FUNCTION_BLOCK _TOD_TestSuite EXTENDS TcUnit.FB_TestSuite
VAR
END_VAR

TestAddress();
TestClearReference();
TestClone();
TestTypeNameReturnsExpected();
TestMakeReferenceToFollowsReference();
TestMakeReferenceToUpdatesReference();
TestSize();
TestValueReturnsExpectedAfterInit();
TestValueReturnsExpectedAfterChange();
TestSerializeTypeWith();
TestSerializeWith();
TestTryDeserializeFrom();
TestTryMakeReferenceToFollowsReference();
TestTryMakeReferenceToUpdatesReference();

METHOD PUBLIC TestAddress
VAR
    _type : _TOD(TOD#0:0:0);
    notExpected : PVOID := 0;
    actual : PVOID;
END_VAR
TEST('TestAddress');

actual := _type.Address;

AssertFalse(
    Condition := (notExpected = actual),
    Message := 'Type did not return a valid address.'
);

TEST_FINISHED();
END_METHOD

METHOD PUBLIC TestClearReference
VAR
    _type : _TOD(TOD#0:0:0);
	target : TOD := TOD#0:0:0;
    expected : TOD := TOD#0:0:0;
    actual : TOD;
END_VAR
TEST('TestClearReference');

_type.MakeReferenceTo(target);
_type.ClearReference();
target := TOD#12:34:56.789;

actual := _type.Value;

AssertEquals(
    Expected := expected,
    Actual := actual,
    Message := 'Value did not follow target change'
);

TEST_FINISHED();
END_METHOD

METHOD PUBLIC TestClone
VAR
    _type : _TIME_OF_DAY(TIME_OF_DAY#12:34:56.789);
	clone : I_Datatype;
	isValidClone : BOOL;
	compareResult : DINT;
END_VAR
TEST('TestClone');

clone := _type.Clone();

isValidClone := clone <> 0;

IF isValidClone THEN
	compareResult := memcmp(_type.Address, clone.Address, clone.Size);
END_IF

AssertTrue(
	Condition := isValidClone,
	Message := 'Clone did not produce a clone'
);

AssertEquals_DINT(
	Expected := 0,
    Actual := compareResult,
    Message := 'Clone did not return a valid clone.'
);

clone.Dispose();

TEST_FINISHED();
END_METHOD

METHOD PUBLIC TestMakeReferenceToFollowsReference
VAR
    _type : _TOD(TOD#0:0:0);
	target : TOD := TOD#0:0:0;
    expected : TOD := TOD#12:34:56.789;
    actual : TOD;
END_VAR
TEST('TestMakeReferenceToFollowsReference');

_type.MakeReferenceTo(target);
target := TOD#12:34:56.789;

actual := _type.Value;

AssertEquals_TIME_OF_DAY(
    Expected := expected,
    Actual := actual,
    Message := 'Value did not follow target change'
);

TEST_FINISHED();
END_METHOD

METHOD PUBLIC TestMakeReferenceToUpdatesReference
VAR
    _type : _TOD(TOD#0:0:0);
	target : TOD := TOD#0:0:0;
    expected : TOD := TOD#12:34:56.789;
    actual : TOD;
END_VAR
TEST('TestMakeReferenceToUpdatesReference');

_type.MakeReferenceTo(target);
_type.Value := TOD#12:34:56.789;

actual := target;

AssertEquals_TIME_OF_DAY(
    Expected := expected,
    Actual := actual,
    Message := 'Value did not update target'
);

TEST_FINISHED();
END_METHOD

METHOD PUBLIC TestSerializeTypeWith
VAR
    _type : _TOD(TOD#0:0:0);
    serializer : JsonSerializer;
    expected : STRING := '{"typeName":"TOD"}';
    actual : STRING(500);
END_VAR
TEST('TestSerializeTypeWith');

serializer.Reset();
_type.SerializeTypeWith(serializer);
serializer.TryGetSerializedData(ADR(actual), SIZEOF(actual));

AssertEquals_STRING(
    Expected := expected,
    Actual := actual,
    Message := 'Serialization of type did not return correct string.'
);

TEST_FINISHED();
END_METHOD

METHOD PUBLIC TestSerializeWith
VAR
    _type : _TOD(TOD#12:34:56.789);
    serializer : JsonSerializer;
    expected : STRING := '"TOD#12:34:56.789"';
    actual : STRING(500);
END_VAR
TEST('TestSerializeWith');

serializer.Reset();
_type.SerializeWith(serializer);
serializer.TryGetSerializedData(ADR(actual), SIZEOF(actual));

AssertEquals_STRING(
    Expected := expected,
    Actual := actual,
    Message := 'Serialization of type data did not return correct string.'
);

TEST_FINISHED();
END_METHOD

METHOD PUBLIC TestSize
VAR
    _type : _TOD(TOD#0:0:0);
    expected : UDINT := SIZEOF(TOD);
    actual : UDINT;
END_VAR
TEST('TestSize');

actual := _type.Size;

AssertEquals_UDINT(
    Expected := Expected,
    Actual := actual,
    Message := 'Type did not return the correct size.'
);

TEST_FINISHED();
END_METHOD

METHOD PUBLIC TestTryDeserializeFrom
VAR
    deserializer : JsonDeserializer;
    feedback : DeserializerFeedback;
    json : STRING := '"TOD#12:34:56.789"';
    _type : _TOD(TOD#0:0:0);
    expected : TOD := TOD#12:34:56.789;
    actual : TOD;
 END_VAR
TEST('TestTryDeserializeFrom');

deserializer.Reset();
deserializer.TryLoad(json);
_type.TryDeserializeFrom(Deserializer, Feedback);

actual := _type.Value;

AssertEquals_TIME_OF_DAY(
    Expected := expected,
    Actual := actual,
    Message := 'Type did not deserialize correctly.'
);

TEST_FINISHED();
END_METHOD

METHOD PUBLIC TestTryMakeReferenceToFollowsReference
VAR
    _type : _TOD(TOD#0:0:0);
	target : _TOD(TOD#0:0:0);
    expected : TOD := TOD#12:34:56.789;
    actual : TOD;
END_VAR
TEST('TestTryMakeReferenceToFollowsReference');

_type.TryMakeReferenceTo(target);
target.Value := TOD#12:34:56.789;

actual := _type.Value;

AssertEquals_TIME_OF_DAY(
    Expected := expected,
    Actual := actual,
    Message := 'Value did not follow target change'
);

TEST_FINISHED();
END_METHOD

METHOD PUBLIC TestTryMakeReferenceToUpdatesReference
VAR
    _type : _TOD(TOD#0:0:0);
	target : _TOD(TOD#0:0:0);
    expected : TOD := TOD#12:34:56.789;
    actual : TOD;
END_VAR
TEST('TestTryMakeReferenceToUpdatesReference');

_type.TryMakeReferenceTo(target);
_type.Value := TOD#12:34:56.789;

actual := target.Value;

AssertEquals_TIME_OF_DAY(
    Expected := expected,
    Actual := actual,
    Message := 'Value did not update target'
);

TEST_FINISHED();
END_METHOD

METHOD PUBLIC TestTypeNameReturnsExpected
VAR
    _type : _TOD(TOD#0:0:0);
    expected : STRING := 'TOD';
    actual : STRING;
END_VAR
TEST('TestTypeNameReturnsExpected');

actual := _type.TypeName;

AssertEquals_STRING(
    Expected := expected,
    Actual := actual,
    Message := 'Type did not return correct iec type.'
);

TEST_FINISHED();
END_METHOD

METHOD PUBLIC TestValueReturnsExpectedAfterChange
VAR
    _type : _TOD(TOD#0:0:0);
    expected : TOD := TOD#12:34:56.789;
    actual : TOD;
END_VAR
TEST('TestValueReturnsExpectedAfterChange');

_type.Value := TOD#12:34:56.789;

actual := _type.Value;

AssertEquals_TIME_OF_DAY(
    Expected := expected,
    Actual := actual,
    Message := 'Expected value not returned after change.'
);

TEST_FINISHED();
END_METHOD

METHOD PUBLIC TestValueReturnsExpectedAfterInit
VAR
    _type : _TOD(TOD#12:34:56.789);
    expected : TOD := TOD#12:34:56.789;
    actual : TOD;
END_VAR
TEST('TestValueReturnsExpectedAfterInit');

actual := _type.Value;

AssertEquals_TIME_OF_DAY(
    Expected := expected,
    Actual := actual,
    Message := 'Expected value not returned after Init.'
);

TEST_FINISHED();
END_METHOD

END_FUNCTION_BLOCK

(* stored: Version 1.1.0.1, ProductVersion 3.1.4024.12
   POU _TOD_TestSuite: Id {19c985da-db57-4090-99b1-9510d3a8ac67}, SpecialFunc None
   Method TestAddress: Id {498e0ce2-8566-4fad-98f3-21d590e725ad}
   Method TestClearReference: Id {1d1ff48f-8829-450a-ba42-080daad2c195}
   Method TestClone: Id {ed9e6f56-b283-41c2-848f-2f760525daff}
   Method TestMakeReferenceToFollowsReference: Id {87f976ac-4356-4c6b-89a1-08f145d30521}
   Method TestMakeReferenceToUpdatesReference: Id {7a1f0d45-26a2-40a1-868b-2ed26d442d56}
   Method TestSerializeTypeWith: Id {efd9c84a-49d7-4b9c-bdef-a0ad39213d16}
   Method TestSerializeWith: Id {653d54dc-973e-4e63-aeca-d1215da6e0b3}
   Method TestSize: Id {1555bde5-6958-4608-9237-c9e6a1148f0b}
   Method TestTryDeserializeFrom: Id {ab34a4d7-88cc-4aee-a8af-b26ac5f1fc37}
   Method TestTryMakeReferenceToFollowsReference: Id {91f7a228-78e5-45d3-8c8a-73245d2536d5}
   Method TestTryMakeReferenceToUpdatesReference: Id {06eb690f-fd88-4eac-98dd-857046fb5cb4}
   Method TestTypeNameReturnsExpected: Id {fd0d099a-5dc5-48c3-9711-671b4a74e988}
   Method TestValueReturnsExpectedAfterChange: Id {3ea3b764-eb54-431e-a750-278087a3657e}
   Method TestValueReturnsExpectedAfterInit: Id {ac6e52c6-eb76-4f61-9a0a-905b2041dd19} *)
